(* IEC 61131-3 sources: CannyIEC/extracted_st/cannyiec/functions/isignbit, 1 file *)

(* ---- ISIGNBIT.st ---- *)
(* --- Interface --- *)
FUNCTION ISIGNBIT : BIT
VAR_INPUT
    iValue : INT;
END_VAR

(* --- Implementation --- *)
ISIGNBIT := iValue < INT#0;
